// TIA Portal V19 export
TYPE "C501_VAR_PMP_TYPIC"
   STRUCT
      STS { ExternalAccessible := 'False'; ExternalVisible := 'False'; ExternalWritable := 'False'} : USInt;   // Status van de pomp
      BMO { ExternalAccessible := 'False'; ExternalVisible := 'False'; ExternalWritable := 'False'} : USInt;   // Bedieningsmode
      BST { ExternalAccessible := 'False'; ExternalVisible := 'False'; ExternalWritable := 'False'} : USInt;   // Bestuurbaarheid
      PWR { ExternalAccessible := 'False'; ExternalVisible := 'False'; ExternalWritable := 'False'} : Real;   // Actueel vermogen van de pomp
      TYD_TOT_AAN { ExternalAccessible := 'False'; ExternalVisible := 'False'; ExternalWritable := 'False'} : LInt;   // Totaal aantal draaiuren
      TYD_AAN { ExternalAccessible := 'False'; ExternalVisible := 'False'; ExternalWritable := 'False'} : Int;   // Tijdsduur dat pomp aangeschakeld is
      TYD_UIT { ExternalAccessible := 'False'; ExternalVisible := 'False'; ExternalWritable := 'False'} : Int;   // Tijdsduur dat pomp uitgeschakeld is
   END_STRUCT;
END_TYPE
